RoboDK station: Kuka_Station1.rdk

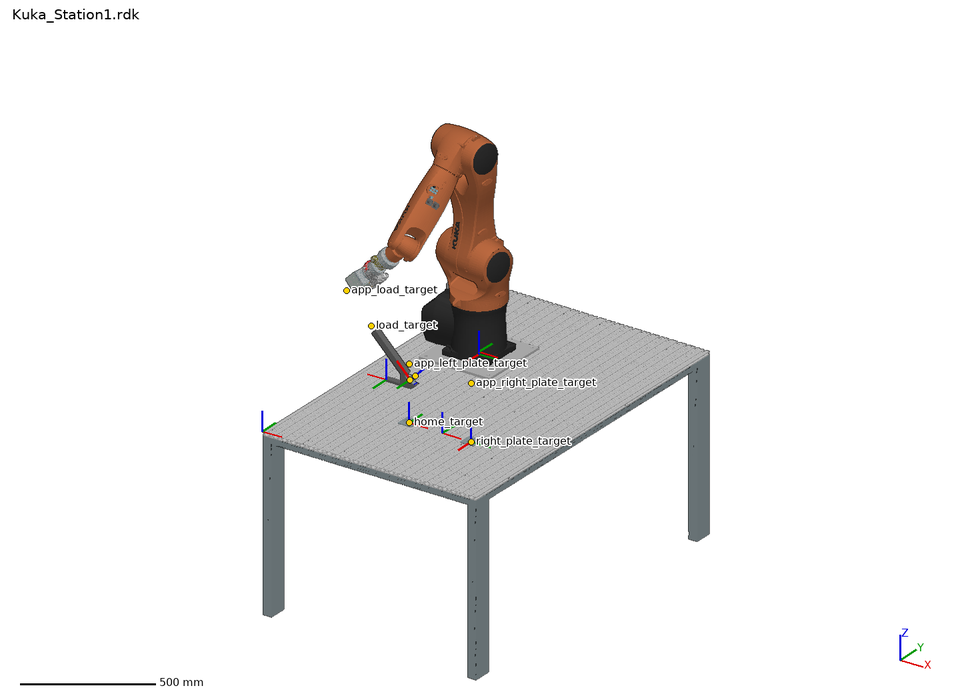
[picture v0: the station drawn from its stored meshes, robots at their saved joint values, targets as dots, program paths as lines]
Station Kuka_Station1 (saved by RoboDK 5.5.2). Poses are relative to the parent item; angles as X-Y-Z fixed-axis rotations.
  - frame table_frame at (0, 0, 0) mm
    - object table_object at (0, 0, 0) mm, size 960.1 x 1500 x 750 mm, geometry from table_object.sld
    - frame base_plate_frame at (280, 990, 0) mm, rotated rx 0 ry 0 rz -90 deg
      - object base_plate_object at (0, 0, 0) mm, size 320 x 320 x 10 mm, geometry from base_plate_object.sld
    - frame slider_frame at (125, 617, 0) mm, rotated rx 0 ry 0 rz 180 deg
      - object slider_object at (0, 0, 0) mm, size 198.7 x 26 x 198.7 mm, 1 curves, geometry from slider_object.sld
    - frame slider_parts_frame at (232.7, 617, 30.7) mm, rotated rx 0 ry -45 rz 180 deg
      - object part_object at (-0.4, 0, -1.01) mm, size 40 x 20 x 20 mm, 1 curves, geometry from part_object.sld
    - frame pick_and_drop_frame at (550, 370, 0) mm
    - frame right_frame at (680, 370, 0) mm, rotated rx 0 ry 0 rz -90 deg
      - object right_plate_object at (0, 0, 0) mm, size 60 x 60 x 9 mm, 1 curves, geometry from right_plate_object.sld
    - frame left_frame at (400, 370, 0) mm
      - object left_plate_object at (0, 0, 0) mm, size 60 x 60 x 9 mm, 1 curves, geometry from left_plate_object.sld
    - frame kuka_frame at (280, 990, 10) mm
      - robot KUKA KR 6 R900 sixx: 6 axes, payload 6 kg, reach 901 mm, repeatability 0.03 mm, weight 52 kg
          modified DH rows (alpha deg, a mm, theta deg, d mm): 0, 0, 0, 400; -90, 25, 0, 0; 0, 455, -90, 0; -90, 35, 0, 420; 90, 0, 0, 0; -90, 0, 180, 80
          joint limits [-170, -190, -120, -185, -120, -350] to [170, 45, 156, 185, 120, 350]; home [0, -90, 90, 0, 0, 0]; saved at [101.131, -84.001, 131.688, 61.605, 52.063, -80.126]
        - robot gripper: 1 axes
            joint limits [0] to [50]; home [0]; saved at [50]
        - tool gripper_TCP, TCP at (0, 0, 288) mm, rotated rx 0 ry 0 rz 43 deg
    - target home_target (Cartesian target) at (399.96, 369.99, -0.03) mm, rotated rx -180 ry 0 rz 0 deg; joints [79.05, -39.88, 97.01, -180, -32.87, 122.05] of KUKA KR 6 R900 sixx
    - target left_plate_target (Cartesian target) at (400, 370, 0) mm, rotated rx -180 ry 0 rz 0 deg; joints [79.046, -39.883, 97.011, -180, -32.872, 122.046] of KUKA KR 6 R900 sixx
    - target app_left_plate_target (Cartesian target) at (400, 370, 240) mm, rotated rx 180 ry 0 rz 0 deg; joints [79.046, -59.338, 91.415, -180, -57.923, 122.046] of KUKA KR 6 R900 sixx
    - target right_plate_target (Cartesian target) at (680, 370, 0) mm, rotated rx 180 ry 0 rz 0 deg; joints [57.171, -30.536, 75.703, -180, -44.833, 100.171] of KUKA KR 6 R900 sixx
    - target app_right_plate_target (Cartesian target) at (680, 370, 240) mm, rotated rx 180 ry 0 rz 0 deg; joints [57.171, -46.58, 69.664, -180, -66.915, 100.171] of KUKA KR 6 R900 sixx
    - target app_slider_parts_target (Cartesian target) at (253.91, 617, 51.91) mm, rotated rx -180 ry 45 rz 0 deg; joints [57.884, -43.74, 126.637, -127.555, -49.065, 50.968] of KUKA KR 6 R900 sixx
    - target slider_parts_target (Cartesian target) at (232.27, 617, 29.7) mm, rotated rx -180 ry 45 rz 0 deg; joints [60.332, -40.77, 127.392, -122.476, -46.744, 47.031] of KUKA KR 6 R900 sixx
    - target load_target (Cartesian target) at (59.33, 616, 202.13) mm, rotated rx -180 ry 45 rz 0 deg; joints [83.964, -69.724, 137.171, 64.204, 51.353, -107.768] of KUKA KR 6 R900 sixx
    - target app_load_target (Cartesian target) at (-53.8, 616, 315.27) mm, rotated rx -180 ry 45 rz 0 deg; joints [101.131, -84.001, 131.688, 61.605, 52.063, -80.126] of KUKA KR 6 R900 sixx
    - target close_gripper_target (joint target) at (-53.8, 616, 315.27) mm, rotated rx -180 ry 45 rz 0 deg; joints [20] of gripper
    - target open_gripper_target (joint target) at (-53.8, 616, 315.27) mm, rotated rx -180 ry 45 rz 0 deg; joints [50] of gripper
    - target Target 12 (Cartesian target) at (-53.8, 616, 315.27) mm, rotated rx -180 ry 45 rz 0 deg; joints [101.131, -84.001, 131.688, 61.605, 52.063, -80.126] of KUKA KR 6 R900 sixx
    - target Target 13 (Cartesian target) at (-53.8, 616, 315.27) mm, rotated rx -180 ry 45 rz 0 deg; joints [101.131, -84.001, 131.688, 61.605, 52.063, -80.126] of KUKA KR 6 R900 sixx
  - folder programs
    - program factory_reset (1 instructions, listed below)
    - program open_gripper (3 instructions, listed below)
    - program close_gripper (3 instructions, listed below)
    - program main (0 instructions, listed below)

--- program factory_reset (robot KUKA KR 6 R900 sixx) ---
  Replace objects

--- program open_gripper (robot gripper) ---
  Set Ref.: table_frame
  Set Tool: gripper_TCP
  MoveJ (Target 12)

--- program close_gripper (robot gripper) ---
  Set Ref.: table_frame
  Set Tool: gripper_TCP
  MoveJ (Target 13)

--- program main ---
